// TIA Portal project "Ejemplo_I" (V16)

(* hardware
DEVICE "PC-System_1"  SIMATIC PC station
   slot 0: "Estación PC SIMATIC"  Rail  SIMATIC PC-Station  V1.0
      slot 125: "Stationmanager"  Station_Manager  V6.0.4
   slot 1: "HMI_RT_1"  WinCC RT Advanced  6AV2 104-0xxxx-xxxx  16.0.0.0
      slot 33792: "Interfaz del equipo"  Host interface
   slot 2: "IE general_1"  IE General  IE_CP  V8.2.0
*)

(* ===== HMI "HMI_RT_1" =====
system functions are stored by id; their names below are inferred from use

HMI tags "Tabla de variables estándar"
   "Texto" : WString[255], internal
   "Sensor_entero" : Int, internal
   "Sensor_real" : Real, internal
   "NombreTabla" : WString[255], internal

screen "Imagen_1" 1024x768
   IOField "Campo ES_1" at 155,18 size 96x32; FormatPattern ???????????????????????????????????????????????????????????????????????????????????????????????????????????????????????????????????????????????????????????????????????????????????????????????????????????????????????????????????????????????????????????????
      ProcessValue <- "Texto"
   Button "Botón_1" at 15,18 size 96x32; TextOff 'Consulta'
      on Click: "Consulta"()
   IOField "Campo ES_2" at 114,89 size 96x32; FormatPattern s99999
      ProcessValue <- "Sensor_entero"
   TextField "Campo de texto_1" at 18,94 size 77x22; Text 'Sensor_1'
   TextField "Campo de texto_2" at 18,150 size 77x22; Text 'Sensor_2'
   IOField "Campo ES_3" at 114,140 size 96x32; FormatPattern s999999999.999
      ProcessValue <- "Sensor_real"
   Button "Botón_2" at 249,88 size 96x32; TextOff 'Insertar'
      on Click: "Insertar"()
   IOField "Campo ES_4" at 15,228 size 110x32; FormatPattern ????????????????????????????????????????????????????????????????????????????????
      ProcessValue <- "NombreTabla"
   TextField "Campo de texto_3" at 15,201 size 109x22; Text 'Nombre Tabla'
   Button "Botón_3" at 155,206 size 96x32; TextOff 'Crear tabla'
      on Click: "Crear"()

VB script "Consulta"
   'Conexiòn y lectura de una BD en SQL
   Dim cn, rs, connectionString, i
   Set cn = CreateObject("ADODB.Connection")
   Set rs = CreateObject("ADODB.Recordset")
   connectionString = "DRIVER={MySQL ODBC 8.0 UNICODE Driver};" & _
    				   "SERVER=localhost:3306;" & _
                      "DATABASE=Procesoautomatica;" & _
                      "UID=root;" & _
                      "PWD=12345;"
   cn.Open connectionString
   rs.Open "SELECT * FROM Tabla1", cn, 3
   rs.MoveFirst
   
   While Not rs.EOF
       SmartTags("Texto")= rs.Fields(0)
       rs.MoveNext
   Wend
   cn.Close

VB script "Insertar"
   'Conexiòn y lectura de una BD en SQL
   Dim cn, rs, connectionString, i
   Set cn = CreateObject("ADODB.Connection")
   Set rs = CreateObject("ADODB.Recordset")
   connectionString = "DRIVER={MySQL ODBC 8.0 UNICODE Driver};" & _
    				   "SERVER=localhost:3306;" & _
                      "DATABASE=Procesoautomatica;" & _
                      "UID=root;" & _
                      "PWD=12345;"
                      
   cn.Open connectionString
   rs.Open "INSERT INTO Tabla1 VALUES(" & SmartTags("Sensor_entero") _
   & "," & SmartTags("Sensor_real") & ");" ,cn, 3
   SmartTags("Texto") = "INSERT INTO Tabla1 VALUES(" _
   & SmartTags("Sensor_entero") & "," & SmartTags("Sensor_real") & ");"
   cn.Close

VB script "Crear"
   'Conexiòn y lectura de una BD en SQL
   Dim cn, rs, connectionString, i
   Set cn = CreateObject("ADODB.Connection")
   Set rs = CreateObject("ADODB.Recordset")
   connectionString = "DRIVER={MySQL ODBC 8.0 UNICODE Driver};" & _
    				   "SERVER=localhost:3306;" & _
                      "DATABASE=Procesoautomatica;" & _
                      "UID=root;" & _
                      "PWD=12345;"
   cn.Open connectionString
   rs.Open "CREATE TABLE " & SmartTags("NombreTabla") _
   & "(ID INT AUTO_INCREMENT PRIMARY KEY, SENSOR_1 INT, SENSOR_2 REAL);" ,cn, 3
   SmartTags("Texto") = "Tabla creada"
   cn.Close
*)